Universal Robots URScript: WORKS.script

def WORKS():
  global _hidden_verificationVariable=0
  set_tool_communication(False, 115200, 0, 1, 1.5, 3.5)
  set_tool_output_mode(0)
  set_tool_digital_output_mode(0, 1)
  set_tool_digital_output_mode(1, 1)
  set_tool_voltage(0)
  set_target_payload(1.000000, [0.000000, 0.000000, 0.000000], [0.001539, 0.001539, 0.001539, 0.000000, 0.000000, 0.000000])
  set_tcp(p[0.0,0.0,0.0,0.0,0.0,0.0])
  set_gravity([0.0, 0.0, 9.82])
  set_safety_mode_transition_hardness(1)
  tool_wrench_limit_disable()
  motion_version_set(2)
  set_standard_analog_input_domain(0, 1)
  set_standard_analog_input_domain(1, 1)
  set_tool_analog_input_domain(0, 1)
  set_tool_analog_input_domain(1, 1)
  set_analog_outputdomain(0, 0)
  set_analog_outputdomain(1, 0)
  set_input_actions_to_default()
  # begin: URCap Installation Node
  #   Source: External Control, 1.0.5, FZI Research Center for Information Technology
  #   Type: External Control
  # end: URCap Installation Node
  step_count_28cebb09_2d9a_42b0_96d3_ddfaf2707272 = 0.0
  thread Step_Counter_Thread_272e11f6_ee2a_4a73_9734_006772467839():
    while (True):
      step_count_28cebb09_2d9a_42b0_96d3_ddfaf2707272 = step_count_28cebb09_2d9a_42b0_96d3_ddfaf2707272 + 1.0
      sync()
    end
  end
  run Step_Counter_Thread_272e11f6_ee2a_4a73_9734_006772467839()
  while (True):
    $ 2 "Robot Program"
    $ 3 "Wait: 1.0"
    sleep(1.0)
    # begin: URCap Program Node
    #   Source: External Control, 1.0.5, FZI Research Center for Information Technology
    #   Type: External Control
    $ 4 "Control by 192.168.56.102"
 # HEADER_BEGIN



 steptime = get_steptime()

 textmsg("ExternalControl: steptime=", steptime)
 MULT_jointstate = 1000000
 MULT_time = 1000

 DEBUG = False

 STOPJ_ACCELERATION = 4.0

 #Constants
 SERVO_UNINITIALIZED = -1
 SERVO_IDLE = 0
 SERVO_RUNNING = 1

 MODE_STOPPED = -2
 MODE_UNINITIALIZED = -1
 MODE_IDLE = 0
 MODE_SERVOJ = 1
 MODE_SPEEDJ = 2
 MODE_FORWARD = 3
 MODE_SPEEDL = 4
 MODE_POSE = 5
 MODE_FREEDRIVE = 6
 MODE_TOOL_IN_CONTACT = 7
 MODE_TORQUE = 8
 # Data dimensions of the message received on the reverse interface
 REVERSE_INTERFACE_DATA_DIMENSION = 8

 TRAJECTORY_MODE_RECEIVE = 1
 TRAJECTORY_MODE_CANCEL = -1

 MOTION_TYPE_MOVEJ = 0
 MOTION_TYPE_MOVEL = 1
 MOTION_TYPE_MOVEP = 2
 MOTION_TYPE_MOVEC = 3
 MOTION_TYPE_OPTIMOVEJ = 4
 MOTION_TYPE_OPTIMOVEL = 5
 MOTION_TYPE_SPLINE = 51
 TRAJECTORY_DATA_DIMENSION = 3 * 6 + 1

 TRAJECTORY_RESULT_SUCCESS = 0
 TRAJECTORY_RESULT_CANCELED = 1
 TRAJECTORY_RESULT_FAILURE = 2

 ZERO_FTSENSOR = 0
 SET_PAYLOAD = 1
 SET_TOOL_VOLTAGE = 2
 START_FORCE_MODE = 3
 END_FORCE_MODE = 4
 START_TOOL_CONTACT = 5
 END_TOOL_CONTACT = 6
 SET_FRICTION_COMPENSATION = 7
 FT_RTDE_INPUT_ENABLE = 8
 SCRIPT_COMMAND_DATA_DIMENSION = 28

 FREEDRIVE_MODE_START = 1
 FREEDRIVE_MODE_STOP = -1

 UNTIL_TOOL_CONTACT_RESULT_SUCCESS = 0
 UNTIL_TOOL_CONTACT_RESULT_CANCELED = 1

 SPLINE_CUBIC = 1
 SPLINE_QUINTIC = 2

 # Maximum allowable joint speed in rad/s
 MAX_JOINT_SPEED = 6.283185

 # Any motion commands resulting in a velocity higher than that will be ignored.
 JOINT_IGNORE_SPEED = 20.0

 #Global variables are also showed in the Teach pendants variable list
 global violation_popup_counter = 0
 global cmd_servo_state = SERVO_UNINITIALIZED
 global cmd_servo_qd = [0.0, 0.0, 0.0, 0.0, 0.0, 0.0]
 global cmd_torque = [0.0, 0.0, 0.0, 0.0, 0.0, 0.0]
 global cmd_servo_q = get_joint_positions()
 global cmd_servo_q_last = cmd_servo_q
 global cmd_twist = [0.0, 0.0, 0.0, 0.0, 0.0, 0.0]
 global extrapolate_count = 0
 global extrapolate_max_count = 0
 global control_mode = MODE_UNINITIALIZED
 global trajectory_points_left = 0
 global spline_qdd = [0, 0, 0, 0, 0, 0]
 global spline_qd = [0, 0, 0, 0, 0, 0]
 global tool_contact_running = False
 global trajectory_result = 0
 global friction_compensation_enabled = True

 # Global thread variables
 thread_move = 0
 thread_trajectory = 0
 thread_script_commands = 0

 ###
 # @brief Function to verify whether the specified target can be reached within the defined time frame while staying within
 # the robot's speed limits
 #
 # @param target array is the joint target to reach
 # @param time float is the time to reach the target
 #
 # @returns bool true if the target is reachable within the robot's speed limits, false otherwise
 ###
 def targetWithinLimits(step_start, step_end, time):
   local idx = 0
   while idx < 6:
     local velocity = norm(step_end[idx] - step_start[idx]) / time
     if velocity > JOINT_IGNORE_SPEED:
       local str = str_cat(
         str_cat("Velocity ", velocity), str_cat(
           str_cat(" required in joint ", idx), str_cat(
             str_cat(" to go from ", step_start[idx]), str_cat(
               str_cat(" to ", step_end[idx]), str_cat(
                 str_cat(" within ", time), " seconds is exceeding the joint velocity limits. Ignoring commands until a valid command is received.")))))
       if violation_popup_counter == 0:
         # We want a popup when an invalid commant is sent. As long as we keep sending invalid
         # commands, we do not want to repeat the popup.
         popup(str, title="External Control speed limit", blocking=False, warning=True)
       end
       if violation_popup_counter * get_steptime() % 5.0 == 0:
         # We want to have a log printed regularly. We are receiving motion commands that are not
         # feasible. The user should have a chance to know about this.
         textmsg(str)
         textmsg("start configuration: ", step_start)
         textmsg("end   configuration: ", step_end)
       end
       violation_popup_counter = violation_popup_counter + 1
       return False
     end
     idx = idx + 1
   end
   if violation_popup_counter > 0:
     textmsg("Received valid command. Resuming execution.")
     violation_popup_counter = 0
   end
   return True
 end

 def trajectory_result_to_str(trajectory_result):
   if trajectory_result == TRAJECTORY_RESULT_SUCCESS:
     return "SUCCESS"
   end
   if trajectory_result == TRAJECTORY_RESULT_CANCELED:
     return "CANCELED"
   end
   if trajectory_result == TRAJECTORY_RESULT_FAILURE:
     return "FAILURE"
   end
   return "UNKNOWN"
 end

 def terminateProgram():
   textmsg("Terminating robot program due to targets sent to the robot is violating robot constraints.")
   stopj(STOPJ_ACCELERATION)
   halt
 end

 def set_servo_setpoint(q):
   cmd_servo_state = SERVO_RUNNING
   if targetWithinLimits(cmd_servo_q, q, steptime):
     cmd_servo_q_last = cmd_servo_q
     cmd_servo_q = q
   # If the target has been interpolating too far away from the robot, so it would trigger the limit
   # check, but the target is close to where the robot currently is, also accept the command.
   # This can, for example, happen if a command series was too fast for the robot to follow, which
   # triggers a path deviation on the commanding side and that is mitigated by a hold-position
   # command.
   elif targetWithinLimits(get_joint_positions(), q, steptime):
     cmd_servo_q_last = cmd_servo_q
     cmd_servo_q = q
   end
 end

 def extrapolate():
   cmd_servo_q_last = cmd_servo_q
   cmd_servo_q = cmd_servo_q + (get_target_joint_speeds() * steptime)
   return cmd_servo_q
 end

 thread servoThread():
   textmsg("ExternalControl: Starting servo thread")
   state = SERVO_IDLE
   while control_mode == MODE_SERVOJ:
     enter_critical
     q = cmd_servo_q
     do_extrapolate = False
     if (cmd_servo_state == SERVO_IDLE):
       do_extrapolate = True
     end
     state = cmd_servo_state
     if cmd_servo_state > SERVO_UNINITIALIZED:
       cmd_servo_state = SERVO_IDLE
     end

     if do_extrapolate:
       extrapolate_count = extrapolate_count + 1
       if extrapolate_count > extrapolate_max_count:
         extrapolate_max_count = extrapolate_count
       end

       q = extrapolate()
       servoj(q, t=steptime, lookahead_time=0.03, gain=2000)

     elif state == SERVO_RUNNING:
       extrapolate_count = 0
       servoj(q, t=steptime, lookahead_time=0.03, gain=2000)
     else:
       extrapolate_count = 0
       sync()
     end
     exit_critical
   end
   textmsg("ExternalControl: servo thread ended")
   stopj(STOPJ_ACCELERATION)
 end

 # Helpers for speed control
 def set_speed(qd):
   cmd_servo_qd = qd
   control_mode = MODE_SPEEDJ
 end

 thread speedThread():
   textmsg("ExternalControl: Starting speed thread")
   while control_mode == MODE_SPEEDJ:
     qd = cmd_servo_qd
     speedj(qd, 40.0, steptime)
   end
   textmsg("ExternalControl: speedj thread ended")
   stopj(STOPJ_ACCELERATION)
 end

 # Helpers for torque control
 def set_torque(target_torque):
   cmd_torque = target_torque
   control_mode = MODE_TORQUE
 end

 thread torqueThread():
   textmsg("ExternalControl: Starting torque thread")
   while control_mode == MODE_TORQUE:
     torque = cmd_torque
     direct_torque(torque, friction_comp=friction_compensation_enabled)
   end
   textmsg("ExternalControl: torque thread ended")
   stopj(STOPJ_ACCELERATION)
 end

 # Function return value (bool) determines whether the robot is moving after this spline segment or
 # not.
 def cubicSplineRun(end_q, end_qd, time, is_last_point=False, is_first_point=False):
   local str = str_cat(end_q, str_cat(end_qd, time))
   textmsg("Cubic spline arg: ", str)

   local start_q = get_joint_positions()
   # Zero time means infinite velocity to reach the target and is therefore impossible
   if time <= 0.0:
     if is_first_point and time == 0.0:
       # If users specify the current joint position with time 0 that may be fine, in that case just
       # ignore that point
       local distance = norm(end_q - start_q)
       if distance < 0.01:
         local splineTimerTraveled = 0.0
         # USED_IN_TEST_SPLINE_INTERPOLATION write_output_float_register(1, splineTimerTraveled)
         textmsg("Ignoring first point with time 0")
         return False
       end
     end
     error_str = "Spline time shouldn't be zero as it would require infinite velocity to reach the target. Canceling motion."
     textmsg(error_str)
     trajectory_result = TRAJECTORY_RESULT_CANCELED
     popup(error_str, title="External Control error", blocking=False, error=True)
     return False
   elif targetWithinLimits(start_q, end_q, time):
     local start_qd = spline_qd

     # Coefficients0 is not included, since we do not need to calculate the position
     local coefficients1 = start_qd
     local coefficients2 = (-3 * start_q + end_q * 3 - start_qd * 2 * time - end_qd * time) / pow(time, 2)
     local coefficients3 = (2 * start_q - 2 * end_q + start_qd * time + end_qd * time) / pow(time, 3)
     local coefficients4 = [0.0, 0.0, 0.0, 0.0, 0.0, 0.0]
     local coefficients5 = [0.0, 0.0, 0.0, 0.0, 0.0, 0.0]
     jointSplineRun(coefficients1, coefficients2, coefficients3, coefficients4, coefficients5, time, is_last_point)
     return True and (is_last_point == False)
   else:
     trajectory_result = TRAJECTORY_RESULT_CANCELED
     return False
   end
 end

 # Function return value (bool) determines whether the robot is moving after this spline segment or
 # not.
 def quinticSplineRun(end_q, end_qd, end_qdd, time, is_last_point=False, is_first_point=False):
   local str = str_cat(end_q, str_cat(end_qd, str_cat(end_qdd, time)))
   textmsg("Quintic spline arg: ", str)

   local start_q = get_joint_positions()
   # Zero time means infinite velocity to reach the target and is therefore impossible
   if time <= 0.0:
     if is_first_point and time == 0.0:
       # If users specify the current joint position with time 0 that may be fine, in that case just
       # ignore that point
       local distance = norm(end_q - start_q)
       if distance < 0.01:
         return False
       end
     end
     error_str = "Spline time shouldn't be zero as it would require infinite velocity to reach the target. Canceling motion."
     textmsg(error_str)
     trajectory_result = TRAJECTORY_RESULT_CANCELED
     popup(error_str, title="External Control error", blocking=False, error=True)
     return False
   elif targetWithinLimits(start_q, end_q, time):
     local start_qd = spline_qd
     local start_qdd = spline_qdd

     # Pre-calculate coefficients
     local TIME2 = pow(time, 2)
     # Coefficients0 is not included, since we do not need to calculate the position
     local coefficients1 = start_qd
     local coefficients2 = 0.5 * start_qdd
     local coefficients3 = (-20.0 * start_q + 20.0 * end_q - 3.0 * start_qdd * TIME2 + end_qdd * TIME2 - 12.0 * start_qd * time - 8.0 * end_qd * time) / (2.0 * pow(time, 3))
     local coefficients4 = (30.0 * start_q - 30.0 * end_q + 3.0 * start_qdd * TIME2 - 2.0 * end_qdd * TIME2 + 16.0 * start_qd * time + 14.0 * end_qd * time) / (2.0 * pow(time, 4))
     local coefficients5 = (-12.0 * start_q + 12.0 * end_q - start_qdd * TIME2 + end_qdd * TIME2 - 6.0 * start_qd * time - 6.0 * end_qd * time) / (2.0 * pow(time, 5))
     jointSplineRun(coefficients1, coefficients2, coefficients3, coefficients4, coefficients5, time, is_last_point)
     return True and (is_last_point == False)
   else:
     trajectory_result = TRAJECTORY_RESULT_CANCELED
     return False
   end
 end

 def jointSplineRun(coefficients1, coefficients2, coefficients3, coefficients4, coefficients5, splineTotalTravelTime, is_last_point):
   # Initialize variables
   local splineTimerTraveled = 0.0
   local scaled_step_time = get_steptime()
   local scaling_factor = 1.0
   local is_slowing_down = False
   local slowing_down_time = 0.0

   # Interpolate the spline in whole time steps
   while (splineTotalTravelTime - splineTimerTraveled) > get_steptime():
     local time_left = splineTotalTravelTime - splineTimerTraveled

     # Maximum deceleration in rad/s^2
     local max_deceleration = 15
     # The time needed to decelerate with 15 rad/s^2 to reach zero velocity when we move at maximum velocity.
     local deceleration_time = MAX_JOINT_SPEED / max_deceleration

     # If the velocity is too large close to the end of the trajectory we scale the
     # trajectory, such that we follow the positional part of the trajectory, but end with zero velocity.
     if (time_left <= deceleration_time) and (is_last_point == True):
       if is_slowing_down == False:

         # Peek what the joint velocities will be if we take a full time step
         local qd = jointSplinePeek(coefficients1, coefficients2, coefficients3, coefficients4, coefficients5, splineTimerTraveled + get_steptime())
         # Compute the time left to decelerate if we take a full time step
         local x = deceleration_time - (time_left - get_steptime())
         is_slowing_down = checkSlowDownRequired(x, qd, max_deceleration)

         if is_slowing_down == True:
           # This will ensure that we scale the trajectory right away
           slowing_down_time = time_left + get_steptime()
           textmsg("Velocity is too fast towards the end of the trajectory. The robot will be slowing down, while following the positional part of the trajectory.")
         end
       end

       if is_slowing_down == True:
         # Compute scaling factor based on time left and total slowing down time
         scaling_factor = time_left / slowing_down_time
         scaled_step_time = get_steptime() * scaling_factor
       end
     end

     splineTimerTraveled = splineTimerTraveled + scaled_step_time
     jointSplineStep(coefficients1, coefficients2, coefficients3, coefficients4, coefficients5, splineTimerTraveled, get_steptime(), scaling_factor, is_slowing_down)
   end

   # Make sure that we approach zero velocity slowly, when slowing down
   if is_slowing_down == True:
     local time_left = splineTotalTravelTime - splineTimerTraveled

     while time_left >= 1e-5:
       time_left = splineTotalTravelTime - splineTimerTraveled
       # Compute scaling factor based on time left and total slowing down time
       scaling_factor = time_left / slowing_down_time
       scaled_step_time = get_steptime() * scaling_factor

       splineTimerTraveled = splineTimerTraveled + scaled_step_time

       jointSplineStep(coefficients1, coefficients2, coefficients3, coefficients4, coefficients5, splineTimerTraveled, get_steptime(), scaling_factor, is_slowing_down)
     end
     scaling_factor = 0.0
   end

   # Last part of the spline which uses less than one time step
   local timeLeftToTravel = splineTotalTravelTime - splineTimerTraveled

   # To round off the float to the steptime step when it is very close to that number (1e-15)
   if timeLeftToTravel == get_steptime():
     timeLeftToTravel = get_steptime()
   end

   jointSplineStep(coefficients1, coefficients2, coefficients3, coefficients4, coefficients5, splineTotalTravelTime, timeLeftToTravel, scaling_factor, is_slowing_down)
 end

 def jointSplineStep(coefficients1, coefficients2, coefficients3, coefficients4, coefficients5, splineTimerTraveled, timestep, scaling_factor, is_slowing_down = False):
   local last_spline_qd = spline_qd
   spline_qd = coefficients1 + 2.0 * splineTimerTraveled * coefficients2 + 3.0 * pow(splineTimerTraveled, 2) * coefficients3 + 4.0 * pow(splineTimerTraveled, 3) * coefficients4 + 5.0 * pow(splineTimerTraveled, 4) * coefficients5
   spline_qdd = 2.0 * coefficients2 + 6.0 * splineTimerTraveled * coefficients3 + 12.0 * pow(splineTimerTraveled, 2) * coefficients4 + 20.0 * pow(splineTimerTraveled, 3) * coefficients5

   spline_qd = spline_qd * scaling_factor

   # Calculate the max needed qdd arg for speedj to distribute the velocity change over the whole timestep no matter the speed slider value
   qdd_max = list_max_norm((spline_qd - last_spline_qd) / timestep)
   # USED_IN_TEST_SPLINE_INTERPOLATION write_output_float_register(1, splineTimerTraveled)
   speedj(spline_qd, qdd_max, timestep)
 end

 # Helper function to see what the velocity will be if we take a full step
 def jointSplinePeek(coefficients1, coefficients2, coefficients3, coefficients4, coefficients5, splineTimerTraveled):
   local qd = coefficients1 + 2.0 * splineTimerTraveled * coefficients2 + 3.0 * pow(splineTimerTraveled, 2) * coefficients3 + 4.0 * pow(splineTimerTraveled, 3) * coefficients4 + 5.0 * pow(splineTimerTraveled, 4) * coefficients5
   return qd
 end


 ###
 # @brief Helper function to figure out if we need to slown down velocity at the last part of the last spline segment.
 #
 # The max_speed and max_deceleration is used to compute a linear velocity profile as function of the time left to decelerate,
 # then we can use the time left to decelerate to find the maximum allowed speed given the time we have left. If we are above
 # the maximum allowed speed, we start slowing down.
 #
 # @param x float is the time left to decelerate
 # @param qd array is the velocity if we take a full step ahead in the spline
 # @param max_deceleration float is the maximum allowed deceleration 15 rad/s^2
 #
 # @returns bool True if slow don is required, false otherwise
 ###
 def checkSlowDownRequired(x, qd, max_deceleration):
   local max_allowable_speed = MAX_JOINT_SPEED - x * max_deceleration
   local idx = 0
   while idx < 6:
     if norm(qd[idx]) > max_allowable_speed:
       return True
     end
     idx = idx + 1
   end
   return False
 end

 ###
 # @brief Find the maximum value in a list the list must be of non-zero length and contain numbers
 # @param list array list
 ###
 def list_max_norm(list):
   # ensure we have something to iterate over
   local length = get_list_length(list)
   if  length < 1:
     popup("Getting the maximum of an empty list is impossible in list_max().", error = True, blocking = True)
     textmsg("Getting the maximum of an empty list is impossible in list_max()")
     halt
   end

   # search for maximum
   local i = 1
   local max = norm(list[0])
   while i < length:
     local tmp = norm(list[i])
     if tmp > max:
       max = tmp
     end
     i = i + 1
   end

   return max
 end

 thread trajectoryThread():
   textmsg("Executing trajectory. Number of points: ", trajectory_points_left)
   local is_first_point = True
   local is_robot_moving = False
   local INDEX_TIME = TRAJECTORY_DATA_DIMENSION
   local INDEX_BLEND = INDEX_TIME + 1
   # same index as blend parameter, depending on point type
   local INDEX_SPLINE_TYPE = INDEX_BLEND
   local INDEX_POINT_TYPE = INDEX_BLEND + 1
   spline_qdd = [0, 0, 0, 0, 0, 0]
   spline_qd = [0, 0, 0, 0, 0, 0]
   enter_critical
   trajectory_result = TRAJECTORY_RESULT_SUCCESS

   while trajectory_result == TRAJECTORY_RESULT_SUCCESS and trajectory_points_left > 0:
     local timeout = 0.5
     if is_robot_moving:
       timeout = get_steptime()
     end
     #reading trajectory point + blend radius + type of point (cartesian/joint based)
     local raw_point = socket_read_binary_integer(TRAJECTORY_DATA_DIMENSION+1+1, "trajectory_socket", timeout)
     trajectory_points_left = trajectory_points_left - 1

     if raw_point[0] > 0:
       local q = [raw_point[1] / MULT_jointstate, raw_point[2] / MULT_jointstate, raw_point[3] / MULT_jointstate, raw_point[4] / MULT_jointstate, raw_point[5] / MULT_jointstate, raw_point[6] / MULT_jointstate]
       local tmptime = raw_point[INDEX_TIME] / MULT_time
       local blend_radius = raw_point[INDEX_BLEND] / MULT_time
       local is_last_point = False
       if trajectory_points_left == 0:
         blend_radius = 0.0
         is_last_point = True
       end
       # MoveJ point
       if raw_point[INDEX_POINT_TYPE] == MOTION_TYPE_MOVEJ:
         acceleration = raw_point[13] / MULT_jointstate
         velocity = raw_point[7] / MULT_jointstate
         movej(q, a = acceleration, v = velocity, t = tmptime, r = blend_radius)

         # reset old acceleration
         spline_qdd = [0, 0, 0, 0, 0, 0]
         spline_qd = [0, 0, 0, 0, 0, 0]

         # Movel point
       elif raw_point[INDEX_POINT_TYPE] == MOTION_TYPE_MOVEL:
         acceleration = raw_point[13] / MULT_jointstate
         velocity = raw_point[7] / MULT_jointstate
         movel(p[q[0], q[1], q[2], q[3], q[4], q[5]], a = acceleration, v = velocity, t = tmptime, r = blend_radius)

         # reset old acceleration
         spline_qdd = [0, 0, 0, 0, 0, 0]
         spline_qd = [0, 0, 0, 0, 0, 0]

       # MoveP point
       elif raw_point[INDEX_POINT_TYPE] == MOTION_TYPE_MOVEP:
         acceleration = raw_point[13] / MULT_jointstate
         velocity = raw_point[7] / MULT_jointstate
         movep(p[q[0], q[1], q[2], q[3], q[4], q[5]], a = acceleration, v = velocity, r = blend_radius)

         # reset old acceleration
         spline_qdd = [0, 0, 0, 0, 0, 0]
         spline_qd = [0, 0, 0, 0, 0, 0]

       elif raw_point[INDEX_POINT_TYPE] == MOTION_TYPE_MOVEC:
         local v = [raw_point[7], raw_point[8], raw_point[9], raw_point[10], raw_point[11], raw_point[12]] / MULT_jointstate
         via = p[v[0], v[1], v[2], v[3], v[4], v[5]]
         target = p[q[0], q[1], q[2], q[3], q[4], q[5]]
         acceleration = raw_point[13] / MULT_jointstate
         velocity = raw_point[14] / MULT_jointstate
         mode = raw_point[15] / MULT_jointstate
         movec(via, target, acceleration, velocity, blend_radius, mode)

         # reset old acceleration
         spline_qdd = [0, 0, 0, 0, 0, 0]
         spline_qd = [0, 0, 0, 0, 0, 0]

       # Joint spline point
       elif raw_point[INDEX_POINT_TYPE] == MOTION_TYPE_SPLINE:

         # Cubic spline
         if raw_point[INDEX_SPLINE_TYPE] == SPLINE_CUBIC:
           qd = [ raw_point[7] / MULT_jointstate, raw_point[8] / MULT_jointstate, raw_point[9] / MULT_jointstate, raw_point[10] / MULT_jointstate, raw_point[11] / MULT_jointstate, raw_point[12] / MULT_jointstate]
           is_robot_moving = cubicSplineRun(q, qd, tmptime, is_last_point, is_first_point)

           # reset old acceleration
           spline_qdd = [0, 0, 0, 0, 0, 0]

           # Quintic spline
         elif raw_point[INDEX_SPLINE_TYPE] == SPLINE_QUINTIC:
           qd = [ raw_point[7] / MULT_jointstate, raw_point[8] / MULT_jointstate, raw_point[9] / MULT_jointstate, raw_point[10] / MULT_jointstate, raw_point[11] / MULT_jointstate, raw_point[12] / MULT_jointstate]
           qdd = [ raw_point[13]/ MULT_jointstate, raw_point[14]/ MULT_jointstate, raw_point[15]/ MULT_jointstate, raw_point[16]/ MULT_jointstate, raw_point[17]/ MULT_jointstate, raw_point[18]/ MULT_jointstate]
           is_robot_moving = quinticSplineRun(q, qd, qdd, tmptime, is_last_point, is_first_point)
         else:
           textmsg("Unknown spline type given:", raw_point[INDEX_POINT_TYPE])
           clear_remaining_trajectory_points()
           trajectory_result = TRAJECTORY_RESULT_FAILURE
         end

       # OptimoveJ point
       elif raw_point[INDEX_POINT_TYPE] == MOTION_TYPE_OPTIMOVEJ:
         acceleration = raw_point[13] / MULT_jointstate
         velocity = raw_point[7] / MULT_jointstate
         optimovej(q, a = acceleration, v = velocity, r = blend_radius)

         if DEBUG:
           textmsg(str_cat("optimovej(", str_cat(
             str_cat("q=", q), str_cat(
               str_cat(", a=", acceleration), str_cat(
                 str_cat(", v=", velocity), str_cat(
                   str_cat(", r=", blend_radius), ")"))))))
         end

         # reset old acceleration
         spline_qdd = [0, 0, 0, 0, 0, 0]
         spline_qd = [0, 0, 0, 0, 0, 0]

       # OptimoveL point
       elif raw_point[INDEX_POINT_TYPE] == MOTION_TYPE_OPTIMOVEL:
         acceleration = raw_point[13] / MULT_jointstate
         velocity = raw_point[7] / MULT_jointstate

         optimovel(p[q[0], q[1], q[2], q[3], q[4], q[5]], a = acceleration, v = velocity, r = blend_radius)

         if DEBUG:
           textmsg(str_cat("optimovel(", str_cat(
             str_cat("q=", p[q[0], q[1], q[2], q[3], q[4], q[5]]), str_cat(
               str_cat(", a=", acceleration), str_cat(
                 str_cat(", v=", velocity), str_cat(
                   str_cat(", r=", blend_radius), ")"))))))
         end

         # reset old acceleration
         spline_qdd = [0, 0, 0, 0, 0, 0]
         spline_qd = [0, 0, 0, 0, 0, 0]
       end
     else:
       textmsg("Receiving trajectory point failed!")
       trajectory_result = TRAJECTORY_RESULT_FAILURE
     end
     is_first_point = False
   end
   exit_critical
   stopj(STOPJ_ACCELERATION)
   socket_send_int(trajectory_result, "trajectory_socket")
   textmsg("Trajectory finished with result ", trajectory_result_to_str(trajectory_result))
 end

 def clear_remaining_trajectory_points():
   while trajectory_points_left > 0:
     raw_point = socket_read_binary_integer(TRAJECTORY_DATA_DIMENSION + 2, "trajectory_socket")
     trajectory_points_left = trajectory_points_left - 1
   end
 end

 # Helpers for speed control
 def set_speedl(twist):
   cmd_twist = twist
   control_mode = MODE_SPEEDL
 end

 thread speedlThread():
   textmsg("Starting speedl thread")
   while control_mode == MODE_SPEEDL:
     twist = cmd_twist
     speedl(twist, 40.0, steptime)
   end
   textmsg("speedl thread ended")
   stopj(STOPJ_ACCELERATION)
 end

 thread servoThreadP():
   textmsg("Starting pose servo thread")
   state = SERVO_IDLE
   while control_mode == MODE_POSE:
     enter_critical
     q = cmd_servo_q
     do_extrapolate = False
     if (cmd_servo_state == SERVO_IDLE):
       do_extrapolate = True
     end
     state = cmd_servo_state
     if cmd_servo_state > SERVO_UNINITIALIZED:
       cmd_servo_state = SERVO_IDLE
     end

     if do_extrapolate:
       extrapolate_count = extrapolate_count + 1
       if extrapolate_count > extrapolate_max_count:
         extrapolate_max_count = extrapolate_count
       end

       q = extrapolate()
       servoj(q, t=steptime, lookahead_time=0.03, gain=2000)

     elif state == SERVO_RUNNING:
       extrapolate_count = 0
       servoj(q, t=steptime, lookahead_time=0.03, gain=2000)
     else:
       extrapolate_count = 0
       sync()
     end
     exit_critical
   end
   textmsg("pose servo thread ended")
   stopj(STOPJ_ACCELERATION)
 end

 def tool_contact_detection():
   # Detect tool contact in the directions that the TCP is moving
   step_back = tool_contact(direction = get_actual_tcp_speed())

   # If tool contact is detected stop movement and move back to intial contact point
   if step_back > 0:
     if control_mode == MODE_FORWARD:
       kill thread_trajectory
       clear_remaining_trajectory_points()
     elif control_mode == MODE_FREEDRIVE:
       textmsg("Leaving freedrive mode")
       end_freedrive_mode()
     else:
       kill thread_move
     end

     # Set control mode to tool in contact, should be cleared by stopping tool contact detection
     control_mode = MODE_TOOL_IN_CONTACT
     stopl(3)

     # Move to initial contact point
     q = get_actual_joint_positions_history(step_back)
     movel(q)
     socket_send_int(UNTIL_TOOL_CONTACT_RESULT_SUCCESS, "script_command_socket")
     textmsg("tool contact detected")
   end
 end

 # Thread to receive one shot script commands, the commands shouldn't be blocking
 thread script_commands():
   while control_mode > MODE_STOPPED:
     raw_command = socket_read_binary_integer(SCRIPT_COMMAND_DATA_DIMENSION, "script_command_socket", 0)
     if raw_command[0] > 0:
       command = raw_command[1]
       if command == ZERO_FTSENSOR:
         zero_ftsensor()
       elif command == SET_PAYLOAD:
         mass = raw_command[2] / MULT_jointstate
         cog = [raw_command[3] / MULT_jointstate, raw_command[4] / MULT_jointstate, raw_command[5] / MULT_jointstate]
         set_payload(mass, cog)
       elif command == SET_TOOL_VOLTAGE:
         tool_voltage = raw_command[2] / MULT_jointstate
         set_tool_voltage(tool_voltage)
       elif command == START_FORCE_MODE:
         task_frame = p[raw_command[2] / MULT_jointstate, raw_command[3] / MULT_jointstate, raw_command[4] / MULT_jointstate, raw_command[5] / MULT_jointstate, raw_command[6] / MULT_jointstate, raw_command[7] / MULT_jointstate]
         selection_vector = [raw_command[8] / MULT_jointstate, raw_command[9] / MULT_jointstate, raw_command[10] / MULT_jointstate, raw_command[11] / MULT_jointstate, raw_command[12] / MULT_jointstate, raw_command[13] / MULT_jointstate]
         wrench = [raw_command[14] / MULT_jointstate, raw_command[15] / MULT_jointstate, raw_command[16] / MULT_jointstate, raw_command[17] / MULT_jointstate, raw_command[18] / MULT_jointstate, raw_command[19] / MULT_jointstate]
         force_type = raw_command[20] / MULT_jointstate
         force_limits = [raw_command[21] / MULT_jointstate, raw_command[22] / MULT_jointstate, raw_command[23] / MULT_jointstate, raw_command[24] / MULT_jointstate, raw_command[25] / MULT_jointstate, raw_command[26] / MULT_jointstate]
         force_mode_set_damping(raw_command[27] / MULT_jointstate)
         # Check whether script is running on CB3 or e-series. Gain scaling can only be set on e-series robots.
         # step time = 0.008: CB3 robot
         # Step time = 0.002: e-series robot
         if (get_steptime() < 0.008):
           force_mode_set_gain_scaling(raw_command[28] / MULT_jointstate)
         end
         force_mode(task_frame, selection_vector, wrench, force_type, force_limits)
       elif command == END_FORCE_MODE:
         end_force_mode()
       elif command == START_TOOL_CONTACT:
         tool_contact_running = True
       elif command == END_TOOL_CONTACT:
         if control_mode != MODE_TOOL_IN_CONTACT:
           # If tool contact hasn't been detected send canceled result
           socket_send_int(UNTIL_TOOL_CONTACT_RESULT_CANCELED, "script_command_socket")
         end
         tool_contact_running = False
       elif command == SET_FRICTION_COMPENSATION:
         if raw_command[2] == 0:
           friction_compensation_enabled = False
         else:
           friction_compensation_enabled = True
         end
       elif command == FT_RTDE_INPUT_ENABLE:
         if raw_command[2] == 0:
           enabled = False
         else:
           enabled = True
         end
         sensor_mass = raw_command[3] / MULT_jointstate
         sensor_offset = [raw_command[4] / MULT_jointstate, raw_command[5] / MULT_jointstate, raw_command[6] / MULT_jointstate]
         sensor_cog = [raw_command[7] / MULT_jointstate, raw_command[8] / MULT_jointstate, raw_command[9] / MULT_jointstate]
         textmsg("calling ft_rtde_input_enable(",
           str_cat(enabled, str_cat(", ",
             str_cat(sensor_mass, str_cat(", ",
               str_cat(to_str(sensor_offset), str_cat(", ",
                 str_cat(to_str(sensor_cog), ")"))))))))
         ft_rtde_input_enable(enabled, sensor_mass, sensor_offset, sensor_cog)
       end
     end
   end
 end

 # HEADER_END

 # NODE_CONTROL_LOOP_BEGINS
 socket_open("192.168.56.102", 50003, "trajectory_socket")
 socket_open("192.168.56.102", 50004, "script_command_socket")
 # This socket should be opened last as it tells the driver when it has control over the robot
 socket_open("192.168.56.102", 50001, "reverse_socket")

 control_mode = MODE_UNINITIALIZED
 thread_move = 0
 thread_trajectory = 0
 trajectory_points_left = 0
 textmsg("ExternalControl: External control active")
 global read_timeout = 0.0 # First read is blocking
 thread_script_commands = run script_commands()
 while control_mode > MODE_STOPPED:
   enter_critical
   params_mult = socket_read_binary_integer(REVERSE_INTERFACE_DATA_DIMENSION, "reverse_socket", read_timeout)
   if params_mult[0] > 0:

     # Convert read timeout from milliseconds to seconds
     read_timeout = params_mult[1] / 1000.0

     if control_mode != params_mult[REVERSE_INTERFACE_DATA_DIMENSION]:
       # Clear remaining trajectory points
       if control_mode == MODE_FORWARD:
         kill thread_trajectory
         if trajectory_points_left > 0:
           clear_remaining_trajectory_points()
           stopj(STOPJ_ACCELERATION)
           socket_send_int(TRAJECTORY_RESULT_CANCELED, "trajectory_socket")
         end
         # Stop freedrive
       elif control_mode == MODE_FREEDRIVE:
         textmsg("Leaving freedrive mode")
         end_freedrive_mode()
       end

       # If tool is in contact, tool contact should be ended before switching control mode
       if control_mode == MODE_TOOL_IN_CONTACT:
         if tool_contact_running == False:
           control_mode = params_mult[REVERSE_INTERFACE_DATA_DIMENSION]
         end
       else:
         control_mode = params_mult[REVERSE_INTERFACE_DATA_DIMENSION]
         join thread_move
       end
       if control_mode == MODE_SERVOJ:
         cmd_servo_q = get_joint_positions()
         thread_move = run servoThread()
       elif control_mode == MODE_SPEEDJ:
         thread_move = run speedThread()
       elif control_mode == MODE_TORQUE:
         thread_move = run torqueThread()
       elif control_mode == MODE_FORWARD:
         kill thread_move
         stopj(STOPJ_ACCELERATION)
       elif control_mode == MODE_SPEEDL:
         thread_move = run speedlThread()
       elif control_mode == MODE_POSE:
         cmd_servo_q = get_joint_positions()
         thread_move = run servoThreadP()
       end
     end

     # Update the motion commands with new parameters
     if control_mode == MODE_SERVOJ:
       q = [params_mult[2] / MULT_jointstate, params_mult[3] / MULT_jointstate, params_mult[4] / MULT_jointstate, params_mult[5] / MULT_jointstate, params_mult[6] / MULT_jointstate, params_mult[7] / MULT_jointstate]
       set_servo_setpoint(q)
     elif control_mode == MODE_SPEEDJ:
       qd = [params_mult[2] / MULT_jointstate, params_mult[3] / MULT_jointstate, params_mult[4] / MULT_jointstate, params_mult[5] / MULT_jointstate, params_mult[6] / MULT_jointstate, params_mult[7] / MULT_jointstate]
       set_speed(qd)
     elif control_mode == MODE_TORQUE:
       torque = [params_mult[2]/ MULT_jointstate, params_mult[3]/ MULT_jointstate, params_mult[4]/ MULT_jointstate, params_mult[5]/ MULT_jointstate, params_mult[6]/ MULT_jointstate, params_mult[7]/ MULT_jointstate]
       set_torque(torque)
     elif control_mode == MODE_FORWARD:
       if params_mult[2] == TRAJECTORY_MODE_RECEIVE:
         kill thread_trajectory
         clear_remaining_trajectory_points()
         trajectory_points_left = params_mult[3]
         thread_trajectory = run trajectoryThread()
       elif params_mult[2] == TRAJECTORY_MODE_CANCEL:
         textmsg("cancel received")
         kill thread_trajectory
         clear_remaining_trajectory_points()
         stopj(STOPJ_ACCELERATION)
         socket_send_int(TRAJECTORY_RESULT_CANCELED, "trajectory_socket")
       end
     elif control_mode == MODE_SPEEDL:
       twist = [params_mult[2] / MULT_jointstate, params_mult[3] / MULT_jointstate, params_mult[4] / MULT_jointstate, params_mult[5] / MULT_jointstate, params_mult[6] / MULT_jointstate, params_mult[7] / MULT_jointstate]
       set_speedl(twist)
     elif control_mode == MODE_POSE:
       pose = p[params_mult[2] / MULT_jointstate, params_mult[3] / MULT_jointstate, params_mult[4] / MULT_jointstate, params_mult[5] / MULT_jointstate, params_mult[6] / MULT_jointstate, params_mult[7] / MULT_jointstate]
       set_servo_setpoint(get_inverse_kin(pose, cmd_servo_q))
     elif control_mode == MODE_FREEDRIVE:
       if params_mult[2] == FREEDRIVE_MODE_START:
         textmsg("Entering freedrive mode")
         freedrive_mode()
       elif params_mult[2] == FREEDRIVE_MODE_STOP:
         textmsg("Leaving freedrive mode")
         end_freedrive_mode()
       end
     end
     # Tool contact is running, but hasn't been detected
     if tool_contact_running == True and control_mode != MODE_TOOL_IN_CONTACT:
       tool_contact_detection()
     end
   else:
     textmsg("Socket timed out waiting for command on reverse_socket. The script will exit now.")
     control_mode = MODE_STOPPED
   end
   exit_critical
 end

 textmsg("ExternalControl: Stopping communication and control")
 join thread_move
 kill thread_trajectory
 kill thread_script_commands
 stopj(STOPJ_ACCELERATION)
 textmsg("ExternalControl: All threads ended")
 socket_close("reverse_socket")
 socket_close("trajectory_socket")
 socket_close("script_command_socket")

 # NODE_CONTROL_LOOP_ENDS
    # end: URCap Program Node
  end
end
